FUNCTION_BLOCK InverseAnalogControl
VAR_INPUT
	
	AnalogInput			:INT; // 150 amps is the max, 32500 bit

END_VAR
VAR_OUTPUT
	
	AnalogOutput		:INT;

END_VAR
VAR

	Holder				:INT ;

END_VAR


Holder := (AnalogInput * -1) + 32767;

IF Holder < 8192 THEN
	
	AnalogOutput := 8192;
ELSE
	
	AnalogOutput := holder;
END_IF

END_FUNCTION_BLOCK

(* stored: Version 1.1.0.1, ProductVersion 3.1.4024.12
   POU InverseAnalogControl: Id {986df66c-529f-477a-9c0e-54b06c140392}, SpecialFunc None *)
